// TwinCAT 3 PLC project CommonLibrary
// ProgramVersion: 3.1.4023.0
// libraries:
//   Tc2_Standard, * (Beckhoff Automation GmbH)
//   Tc2_System, * (Beckhoff Automation GmbH)
// project tree:
//   HMI/Button/DUTs/ E_Hmi_ButtonBehaviour.TcDUT (not stored), S_Hmi_Button.TcDUT
//   HMI/Button/ FB_Hmi_Button.TcPOU
//   HMI/ FB_Hmi_Component.TcPOU
//   HMI/Led/DUTs/ E_Hmi_LedColor.TcDUT (not stored), S_Hmi_Led.TcDUT (not stored)
//   HMI/Led/ FB_Hmi_Led.TcPOU
//   HMI/Switch/DUTs/ S_Hmi_Switch.TcDUT
//   HMI/Switch/ FB_Hmi_Switch.TcPOU
//   Utilities/DUTs/ LoopIterator.TcDUT (not stored)
//   Utilities/GVLs/ GENERAL.TcGVL
//   Utilities/InitializeControl/ ASSERT.TcPOU, FB_InitializeControl.TcPOU
//   Utilities/InitializeControl/GVLs/ INITIALIZE.TcGVL (not stored)
//   Utilities/MessageHandler/DUTs/ E_Msg_Acknowledge.TcDUT, E_Msg_Behaviour.TcDUT (not stored), E_Msg_Option.TcDUT, S_Msg_Message.TcDUT
//   Utilities/MessageHandler/ FB_MessageHandler.TcPOU
//   Utilities/MessageHandler/GVLs/ MSG.TcGVL (not stored)
//   Utilities/Timers/ FB_Timer.TcPOU, FB_TimerManager.TcPOU, I_Timer.TcIO
//   Utilities/Timers/GVLs/ TIMERS.TcGVL (not stored)

// ---- HMI/Button/DUTs/S_Hmi_Button.TcDUT
TYPE S_Hmi_Button :
STRUCT
	Click: BOOL;
	Enabled: BOOL;
	Visibility: BOOL;
	Value: BOOL;
	Led: S_Hmi_Led;
END_STRUCT
END_TYPE

// ---- HMI/Switch/DUTs/S_Hmi_Switch.TcDUT
TYPE S_Hmi_Switch :
STRUCT
	Click: BOOL;
	Enabled: BOOL;
	Visibility: BOOL;
	Value: BOOL;
END_STRUCT
END_TYPE

// ---- Utilities/MessageHandler/DUTs/E_Msg_Acknowledge.TcDUT
{attribute 'qualified_only'}
{attribute 'strict'}
TYPE E_Msg_Acknowledge :
(
	ByOperator := 0,
	Auto := 1
)UINT;
END_TYPE

// ---- Utilities/MessageHandler/DUTs/E_Msg_Option.TcDUT
{attribute 'qualified_only'}
{attribute 'strict'}
TYPE E_Msg_Option :
(
	None := 0,
	OneParam := 1,
	TwoParam := 2
)UINT;
END_TYPE

// ---- Utilities/MessageHandler/DUTs/S_Msg_Message.TcDUT
TYPE S_Msg_Message :
STRUCT
	Section: UINT;
	Id: UINT;
	Behaviour: E_Msg_Behaviour;
	Option: E_Msg_Option;
	Param_1: STRING;
	Param_2: STRING;
END_STRUCT
END_TYPE

// ---- Utilities/GVLs/GENERAL.TcGVL
VAR_GLOBAL CONSTANT
	MAX_STRING_LENGTH: INT := 255;
ENd_VAR

// ---- Utilities/Timers/I_Timer.TcIO
INTERFACE I_Timer

METHOD Execute
END_METHOD

METHOD Register : BOOL
END_METHOD

END_INTERFACE

// ---- HMI/Button/FB_Hmi_Button.TcPOU
FUNCTION_BLOCK FB_Hmi_Button EXTENDS FB_Hmi_Component
VAR
	_rButton: REFERENCE TO S_Hmi_Button;

	_Led: FB_Hmi_Led;

	_behaviour: E_Hmi_ButtonBehaviour;
END_VAR

IF _initialized THEN
	IF _behaviour = E_Hmi_ButtonBehaviour.MomentaryOff THEN
		_rButton.Value := TRUE;
	ELSIF _behaviour = E_Hmi_ButtonBehaviour.MomentaryOn THEN
		_rButton.Value := FALSE;
	END_IF

	IF _rButton.Click THEN
		CASE _behaviour OF
			E_Hmi_ButtonBehaviour.MomentaryOff:
				Reset();

			E_Hmi_ButtonBehaviour.MomentaryOn:
				Set();

			E_Hmi_ButtonBehaviour.Reset:
				Reset();

			E_Hmi_ButtonBehaviour.Set:
				Set();

			E_Hmi_ButtonBehaviour.Toggle:
				Toggle();
		END_CASE
	END_IF
END_IF

_rButton.Click := FALSE;

PROPERTY PUBLIC Enabled : BOOL
SET
_rButton.Enabled := Enabled;
END_SET
END_PROPERTY

METHOD PUBLIC Initialize : BOOL
VAR_INPUT
	rButton: REFERENCE TO S_Hmi_Button;
	behaviour: E_Hmi_ButtonBehaviour;
END_VAR
IF __ISVALIDREF(rButton) THEN
	_Led.initialize(rButton.Led);
	_rButton REF= rButton;
	_behaviour := behaviour;

	_initialized := Initialize := TRUE;
END_IF
END_METHOD

PROPERTY PUBLIC Led : POINTER TO FB_Hmi_Led;
GET
Led := ADR(_Led);
END_GET
END_PROPERTY

METHOD PUBLIC Reset
IF _initialized AND_THEN _rButton.Enabled THEN
	_rButton.Value := FALSE;
END_IF
END_METHOD

METHOD PUBLIC Set
IF _initialized AND_THEN _rButton.Enabled THEN
	_rButton.Value := TRUE;
END_IF
END_METHOD

METHOD PUBLIC Toggle
IF _initialized AND_THEN _rButton.Enabled THEN
	_rButton.Value := NOT _rButton.Value;
END_IF
END_METHOD

PROPERTY PUBLIC Value : BOOL
GET
Value := _rButton.Value;
END_GET
END_PROPERTY

PROPERTY PUBLIC Visibility : BOOL
SET
IF _initialized THEN
	_rButton.Visibility := Visibility;
END_IF
END_SET
END_PROPERTY

END_FUNCTION_BLOCK

// ---- HMI/FB_Hmi_Component.TcPOU
FUNCTION_BLOCK ABSTRACT FB_Hmi_Component
VAR
	_initialized: BOOL;
END_VAR

PROPERTY PUBLIC ABSTRACT Visibility : BOOL
SET
END_SET
END_PROPERTY

END_FUNCTION_BLOCK

// ---- HMI/Led/FB_Hmi_Led.TcPOU
FUNCTION_BLOCK FB_Hmi_Led EXTENDS FB_Hmi_Component
VAR
	_rLed: REFERENCE TO S_Hmi_Led;

	_blink: BOOL;
	_blinkTime: TIME;
	_Blinker: FB_Timer;
END_VAR

IF _blink THEN
	IF _Blinker.Done THEN
		_Blinker.Start(_blinkTime);
		_rLed.OnOff := NOT _rLed.OnOff;
	END_IF
END_IF

PROPERTY PUBLIC Blink : BOOL
SET
_blink := Blink;
_rLed.OnOff := FALSE;
END_SET
END_PROPERTY

PROPERTY PUBLIC BlinkTime : TIME
SET
BlinkTime := _blinkTime;
END_SET
END_PROPERTY

METHOD PUBLIC Initialize : BOOL
VAR_INPUT
	rLed: REFERENCE TO S_Hmi_Led;
END_VAR
IF __ISVALIDREF(rLed) THEN
	_rLed REF= rLed;
	_initialized := Initialize := TRUE;
END_IF
END_METHOD

PROPERTY PUBLIC OffColor : UINT
SET
_rLed.OffColor := OffColor;
END_SET
END_PROPERTY

PROPERTY PUBLIC OnColor : UINT
SET
_rLed.OnColor := OnColor;
END_SET
END_PROPERTY

PROPERTY PUBLIC OnOff : BOOL
SET
_rLed.OnOff := OnOff;
END_SET
END_PROPERTY

PROPERTY PUBLIC Visibility : BOOL
SET
_rLed.Visibility := Visibility;
END_SET
END_PROPERTY

END_FUNCTION_BLOCK

// ---- Utilities/Timers/FB_Timer.TcPOU
FUNCTION_BLOCK FB_Timer IMPLEMENTS I_Timer
VAR
	_Timer: TON;

	_done: BOOL;
	_busy: BOOL;
	_free: BOOL := TRUE;
END_VAR

PROPERTY PUBLIC Busy : BOOL
GET
Busy := _busy;
END_GET
END_PROPERTY

PROPERTY PUBLIC Done : BOOL
GET
Done := _done;
END_GET
END_PROPERTY

PROPERTY PUBLIC ElapsedTime : TIME
GET
ElapsedTime := _Timer.ET;
END_GET
END_PROPERTY

METHOD Execute
_Timer();

IF _Timer.Q THEN
	_done := TRUE;
	_busy := FALSE;
END_IF
END_METHOD

METHOD Register : BOOL
Register := TIMERS.Manager.Register(THIS^);
END_METHOD

METHOD PUBLIC Reset
_Timer(IN := FALSE);

_done := FALSE;
_busy := FALSE;
_free := TRUE;
END_METHOD

METHOD PUBLIC Start
VAR_INPUT
	delay: TIME;
END_VAR
IF _free THEN
	_Timer(IN := FALSE);
	_Timer(IN := TRUE,
			PT := delay);

	_busy := TRUE;
	_done := FALSE;
	_free := FALSE;
END_IF
END_METHOD

END_FUNCTION_BLOCK

// ---- HMI/Switch/FB_Hmi_Switch.TcPOU
FUNCTION_BLOCK FB_Hmi_Switch EXTENDS FB_Hmi_Component
VAR
	_rSwitch: REFERENCE TO S_Hmi_Switch;
END_VAR

IF _initialized THEN
	IF _rSwitch.Click THEN
		Toggle();
	END_IF
END_IF

_rSwitch.Click := FALSE;

PROPERTY PUBLIC Enabled : BOOL
SET
_rSwitch.Enabled := Enabled;
END_SET
END_PROPERTY

METHOD PUBLIC Initialize : BOOL
VAR_INPUT
	rSwitch: REFERENCE TO S_Hmi_Switch;
END_VAR
IF __ISVALIDREF(rSwitch) THEN
	_rSwitch REF= rSwitch;

	_initialized := Initialize := TRUE;
END_IF
END_METHOD

METHOD PUBLIC Reset
IF _initialized AND_THEN _rSwitch.Enabled THEN
	_rSwitch.Value := FALSE;
END_IF
END_METHOD

METHOD PUBLIC Set
IF _initialized AND_THEN _rSwitch.Enabled THEN
	_rSwitch.Value := TRUE;
END_IF
END_METHOD

METHOD PUBLIC Toggle
IF _initialized AND_THEN _rSwitch.Enabled THEN
	_rSwitch.Value := NOT _rSwitch.Value;
END_IF
END_METHOD

PROPERTY PUBLIC Value : BOOL
GET
Value := _rSwitch.Value;
END_GET
END_PROPERTY

PROPERTY PUBLIC Visibility : BOOL
SET
IF _initialized THEN
	_rSwitch.Visibility := Visibility;
END_IF
END_SET
END_PROPERTY

END_FUNCTION_BLOCK

// ---- Utilities/InitializeControl/ASSERT.TcPOU
FUNCTION ASSERT : BOOL
VAR_INPUT
	passed: BOOL;
	text: STRING;
END_VAR
VAR
END_VAR

IF NOT passed THEN
	ADSLOGSTR(msgCtrlMask := ADSLOG_MSGTYPE_ERROR, msgFmtStr := 'FAILED: %s', text);
END_IF

ASSERT := passed;

END_FUNCTION

// ---- Utilities/InitializeControl/FB_InitializeControl.TcPOU
FUNCTION_BLOCK FB_InitializeControl
VAR
	_passed: BOOL;
	_initList: ARRAY [1..INITIALIZE.MAX_INIT_LIST] OF BOOL;
	_headerText: STRING;
	_totalCounter: INT;
	_passedCounter: INT;
	_failedCounter: INT;
END_VAR

METHOD Footer
ADSLOGSTR(msgCtrlMask := ADSLOG_MSGTYPE_ERROR, msgFmtStr := 'Total Tests: %s', TO_STRING(_totalCounter));
ADSLOGSTR(msgCtrlMask := ADSLOG_MSGTYPE_ERROR, msgFmtStr := 'Passed: %s', TO_STRING(_passedCounter));
ADSLOGSTR(msgCtrlMask := ADSLOG_MSGTYPE_ERROR, msgFmtStr := 'Failed: %s', TO_STRING(_failedCounter));
END_METHOD

METHOD Header
VAR_INPUT
	title: STRING;
END_VAR
_headerText := CONCAT('==========', title);
_headerText := CONCAT(_headerText, ' INITIALIZING==========');

ADSLOGSTR(ADSLOG_MSGTYPE_ERROR, _headerText, '');
END_METHOD

PROPERTY Passed : BOOL
GET
Passed := _passed;
END_GET
SET
IF _totalCounter >= MAX_INIT_LIST THEN
	RETURN;
END_IF

_totalCounter := _totalCounter + 1;

IF Passed THEN
	_passedCounter := _passedCounter + 1;
ELSE
	_failedCounter := _failedCounter + 1;
END_IF

_initList[_totalCounter] := Passed;

_passed := Passed AND _passed;
END_SET
END_PROPERTY

END_FUNCTION_BLOCK

// ---- Utilities/MessageHandler/FB_MessageHandler.TcPOU
FUNCTION_BLOCK FB_MessageHandler
VAR_INPUT
END_VAR
VAR_OUTPUT
END_VAR
VAR
END_VAR

METHOD m_AddStringParam : BOOL
VAR_INPUT
	text: REFERENCE TO T_MaxString;
	param: STRING;
END_VAR
VAR
	_iter: LoopIterator;

	_length: INT;
	_index: INT;
END_VAR
_length := LEN(text) - 2;
_length := _length + LEN(param);


IF ASSERT(_length > MAX_STRING_LENGTH, CONCAT('FB_TimerManager: Maximum amount of timer has ben exceeded - ', TO_STRING(_count + 1))) THEN
	RETURN;
END_IF

FOR _iter := 0 TO LEN(text) DO
	IF text[_iter] = '%' AND text[_iter + 1] = 'S' THEN
		_index := _iter;
		EXIT;
	END_IF
END_FOR

text := REPLACE(text, param, 2, _index);
END_METHOD

METHOD Report : BOOL
VAR_INPUT
END_VAR
END_METHOD

END_FUNCTION_BLOCK

// ---- Utilities/Timers/FB_TimerManager.TcPOU
FUNCTION_BLOCK FB_TimerManager
VAR
	_aTimers: ARRAY [1..TIMERS.MAX_TIMER] OF I_Timer;
	_count: INT := 1;

	_timerIter: LoopIterator;
END_VAR

FOR _timerIter := 1 TO _count DO
	_aTimers[_timerIter].Execute();
END_FOR

METHOD PUBLIC Register : BOOL
VAR_INPUT
	iTimer: I_Timer;
END_VAR
IF ASSERT(iTimer <> 0, CONCAT('FB_TimerManager: Invalid iTimer - ', TO_STRING(_count))) THEN
	IF ASSERT(_count < TIMERS.MAX_TIMER, CONCAT('FB_TimerManager: Maximum amount of timer has ben exceeded - ', TO_STRING(_count + 1))) THEN
		_count := _count + 1;
		_aTimers[_count] := iTimer;
		Register := TRUE;
	END_IF
END_IF
END_METHOD

END_FUNCTION_BLOCK
